FUNCTION_BLOCK DistStnPusher (* Basic Function Block Type *)
  (* Standard: 61499-2 *)
  (* Version 0.2, 2003-12-04, JHC, Rockwell Automation, Renamed for better indexing. *)
  (* Compiler header: package fb.rt.wago; #include <sys/time.h> *)
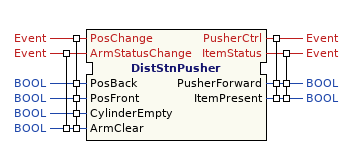
  EVENT_INPUT
    PosChange WITH PosBack, PosFront, CylinderEmpty, ArmClear; (* Normal Execution Request *)
    ArmStatusChange WITH ArmClear;
  END_EVENT
  EVENT_OUTPUT
    PusherCtrl WITH PusherForward, ItemPresent;
    ItemStatus WITH PusherForward, ItemPresent; (* Execution Confirmation *)
  END_EVENT
  VAR_INPUT
    PosBack : BOOL := false; (* Input event qualifier *)
    PosFront : BOOL := false; (* Input event qualifier *)
    CylinderEmpty : BOOL := false; (* Input event qualifier *)
    ArmClear : BOOL;
  END_VAR
  VAR_OUTPUT
    PusherForward : BOOL := false;
    ItemPresent : BOOL := false; (* Output event qualifier *)
  END_VAR
  VAR
    pusherTimer : DATE_AND_TIME;
    timeout : BOOL := false;
  END_VAR
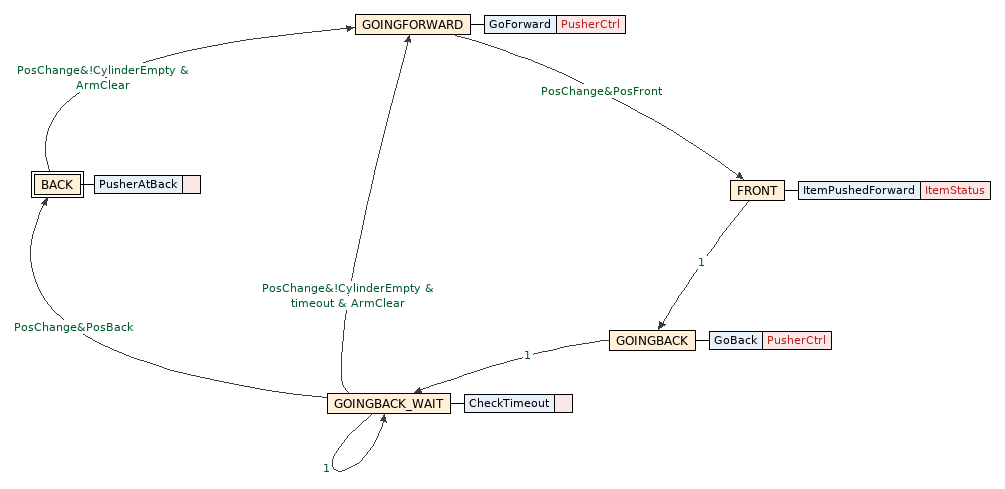
  EC_STATES
    BACK : PusherAtBack; (* Initial State *)
    GOINGBACK : GoBack -> PusherCtrl; (* Normal execution *)
    GOINGBACK_WAIT : CheckTimeout; (* Normal execution *)
    GOINGFORWARD : GoForward -> PusherCtrl;
    FRONT : ItemPushedForward -> ItemStatus;
  END_STATES
  EC_TRANSITIONS
    BACK TO GOINGFORWARD := PosChange&!CylinderEmpty & ArmClear;
    GOINGFORWARD TO FRONT := PosChange&PosFront;
    FRONT TO GOINGBACK := 1;
    GOINGBACK TO GOINGBACK_WAIT := 1;
    GOINGBACK_WAIT TO BACK := PosChange&PosBack;
    GOINGBACK_WAIT TO GOINGFORWARD := PosChange&!CylinderEmpty & timeout & ArmClear;
    GOINGBACK_WAIT TO GOINGBACK_WAIT := 1;
  END_TRANSITIONS
  ALGORITHM GoBack IN C: (* Initialization algorithm *)
me->PusherForward = false;
me->timeout = false;
gettimeofday(&(me->pusherTimer), NULL);
  END_ALGORITHM
  ALGORITHM GoForward IN C: (* Initialization algorithm *)
me->PusherForward = true;
  END_ALGORITHM
  ALGORITHM ItemPushedForward IN C: (* Normally executed algorithm *)
me->ItemPresent = true;
  END_ALGORITHM
  ALGORITHM CheckTimeout IN C:
struct timeval nowtime, timediff;
long long result;

gettimeofday(&nowtime, NULL);
timersub(&nowtime, &me->pusherTimer, &timediff);
result = (long long)(timediff.tv_sec) * 1000000 + timediff.tv_usec;
if( result > 5000000 )
me->timeout = true;
  END_ALGORITHM
END_FUNCTION_BLOCK
